PROGRAM MAIN
VAR
	timer : FB_TIMER();
	trigger : BOOL;
	busy: BOOL;
	errorID_sdo: UDINT;
	sdo_ret_value : UDINT;
	
	check_for_error : BOOL := FALSE;
	reset_drive: BOOL;
	fbSdoRead       : FB_EcCoESdoRead;
	error : BOOL;
	
	state : UINT := 0;
	
	bStatusEnable : BOOL;
		// =============== Axis reference =========================
	AxisRef			: AXIS_REF;				// Axis reference (process data plc/nc)
	
	// =============== Motion function blocks =================
	fbMcPower 		: MC_Power;				// FB for enable and override
	fbMcReset 		: MC_Reset;				// FB to reset axis
	
	// Signal generator
	fbSignalGenerator : FB_CTRL_SIGNAL_GENERATOR;
	fManValue : REAL := 0;
	eMode : E_CTRL_MODE := eCTRL_MODE_ACTIVE;
	stParams : ST_CTRL_SIGNAL_GENERATOR_PARAMS;
	fOut : LREAL;
END_VAR

(*
Change in GVL (GVLs->GVL): 
	TARGET_AMPLITUDE_VELOCITY : DINT := 1000;
	SINUS_FREQUENCY : TIME := T#300MS; // Milliseconds
	AMPLITUDE_OFFSET : REAL := 0.0;

	RESET_HOLD_TIME : TIME := T#2S;
	RESET_SIGNAL : TIME := T#10S;
*)



CASE state OF
	0:
		// Init state
		fbMCPower(	Enable 			:= TRUE, 
			Enable_Positive	:= TRUE, 
			Enable_Negative	:= TRUE, 
			Override		:= 100.0,
			Axis			:= AxisRef,
			Status			=> bStatusEnable);
			
		stParams.eSignalType := eCTRL_SINUS;
		stParams.fAmplitude := GVL.TARGET_AMPLITUDE;
		stParams.fOffset := GVL.AMPLITUDE_OFFSET;
		stParams.tStart := T#0S;
		stParams.tCtrlCycleTime := T#1MS;
		stParams.tTaskCycleTime := T#1MS;
		stParams.tCylceDuration := GVL.SINUS_FREQUENCY; 
		state := 1;
	
	1:
		// Execute state
		// Signal generator for velocity. 
		stParams.fAmplitude := GVL.TARGET_AMPLITUDE;
		fbSignalGenerator(fManValue := fManValue, eMode := eMode, fOut => fOut, stParams := stParams);
		GVL.velocity_out := LREAL_TO_DINT(fOut);
		GVL.torque_out := LREAL_TO_INT(fOut);
		IF eMode = eCTRL_MODE_RESET THEN
			eMode := eCTRL_MODE_ACTIVE;
		END_IF
	
		// Timer for error checking
		timer(trigger => trigger);
		
		IF trigger THEN
			check_for_error := TRUE;
		END_IF
		
		IF check_for_error THEN
			
			// Read SDO Error Object
			fbSDORead(sNetId := GVL.NET_ID_CABINET,
					nSlaveAddr := GVL.SLAVE_ADDR, 
					nIndex := GVL.OBJ_DIR_ERROR, 
					nSubIndex := 0, 
					pDstBuf := ADR(sdo_ret_value), 
					cbBuflen := SIZEOF(sdo_ret_value), 
					bExecute := TRUE, 
					bError => error, 
					nErrId => errorID_sdo, 
					bBusy => busy);
			// If error value unequal zero, reset drive.		
			IF sdo_ret_value <> 0 THEN
				reset_drive := TRUE;
				// Reset signal generator
				eMode := eCTRL_MODE_RESET;					
			END_IF
				// Finish SDO Reading
				fbSDORead(sNetId := GVL.NET_ID_CABINET,
					nSlaveAddr := GVL.SLAVE_ADDR, 
					nIndex := GVL.OBJ_DIR_ERROR, 
					nSubIndex := 0, 
					pDstBuf := ADR(sdo_ret_value), 
					cbBuflen := SIZEOF(sdo_ret_value), 
					bExecute := FALSE, 
					bError => error, 
					nErrId => errorID_sdo, 
					bBusy => busy);
			check_for_error := FALSE;
		END_IF
		
		// Call reset functions
		// Reset Drive
		F_DRIVE_RESET(reset_drive);
		// Reset NC Task
		fbMcReset(Execute := reset_drive, Axis := AxisRef);
		reset_drive := FALSE;
END_CASE

END_PROGRAM

(* stored: Version 1.1.0.1, ProductVersion 3.1.4022.16
   POU MAIN: Id {6e890035-cf79-4130-96a8-f7c09ccea42f}, SpecialFunc None *)
